FUNCTION_BLOCK PtPreciseDiff
VAR_INPUT
	years: DINT;
    months: DINT;
    days: DINT;
    hours: DINT;
    minutes: DINT;
    seconds: DINT;
    microseconds: DINT;
    total_days: DINT;
END_VAR
VAR_OUTPUT
END_VAR
VAR
END_VAR

METHOD Set : BOOL
VAR_INPUT
	years: DINT;
    months: DINT;
    days: DINT;
    hours: DINT;
    minutes: DINT;
    seconds: DINT;
    microseconds: DINT;
    total_days: DINT;
END_VAR
THIS^.years := years;
THIS^.months := months;
THIS^.days := days;
THIS^.hours := hours;
THIS^.minutes := minutes;
THIS^.seconds := seconds;
THIS^.microseconds := microseconds;
THIS^.total_days := total_days;
END_METHOD

END_FUNCTION_BLOCK

(* stored: Version 1.1.0.1, ProductVersion 3.1.4024.12
   POU PtPreciseDiff: Id {712dc1f4-25ad-4265-8045-422cc0d0a301}, SpecialFunc None
   Method Set: Id {7fa07a64-4ba5-4fbf-9d05-7af5a915a08d} *)
